INTERFACE ITF_State

METHOD Cycle : BOOL
VAR_INPUT
END_VAR
END_METHOD

END_INTERFACE

(* stored: Version 1.1.0.1, ProductVersion 3.1.4024.12
   Itf ITF_State: Id {0083945d-138d-4ad6-9991-4b6d9f0ab67c}
   Method Cycle: Id {88ffa559-518d-46cc-8f55-5c56294c1a45} *)
